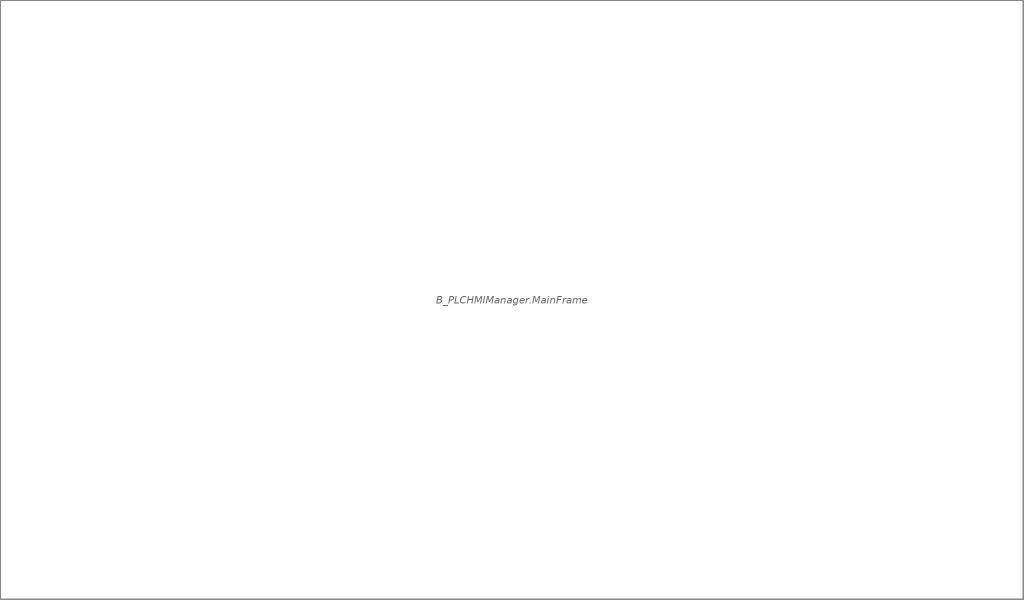
VISUALIZATION MainScreen  // 1024x600
    Frame (0,0 1024x600)
        shows B_PLCHMIManager.MainFrame(stHMIData := PRG_ControlHMI.stHMIData)
END_VISUALIZATION

(* stored: Version 1.1.0.1, ProductVersion 3.1.4024.15
   Visu MainScreen: Id {3c5eb390-ca10-415d-b24b-5a44a6258059} *)
